PROGRAM MAIN
VAR
	startButton : StartButton;
END_VAR

startButton();

END_PROGRAM

(* stored: Version 1.1.0.1, ProductVersion 3.1.4024.12
   POU MAIN: Id {15b7f900-a103-4422-886a-9998b8f48822}, SpecialFunc None *)
